// TIA Portal V17 export
// export: Created 2022-07-20T07:01:33.4482737Z, ExportSetting WithDefaults, DisplayName Totally Integrated Automation Portal, DisplayVersion V17, DisplayName TIA Portal Openness, DisplayVersion V17, DisplayName TIA Portal Version Control Interface, DisplayVersion V17, DisplayName SINAMICS Startdrive Advanced, DisplayVersion V17, DisplayName SINAMICS Startdrive G130, G150, S120, S150, SINAMICS MV, S210, DisplayVersion V17, DisplayName SINAMICS Startdrive G110M, G120, G120C, G120D, G120P, G115D, DisplayVersion V17, DisplayName STEP 7 Professional, DisplayVersion V17, DisplayName STEP 7 Safety, DisplayVersion V17, DisplayName WinCC Advanced, DisplayVersion V17
FUNCTION_BLOCK "FB10322_PrinterCompactInkCircuit"   // FB10322, LAD
{ S7_Optimized_Access := 'TRUE' }
VERSION : 0.1
// stored: AutoNumber false, IsIECCheckEnabled false, IsRetainMemResEnabled false, MemoryReserve 100, SetENOAutomatically false, UDAEnableTagReadback false
   VAR_INPUT
      InkWeighScale_RawValue : Int;
      InkWeighScale_CalibrationValue_1 : Real;
      InkWeighScale_CalibrationValue_2 : Real;
      InkWeighScale_HighErrorThreshold : Real;
      InkWeighScale_HighWarningThreshold : Real;
      InkWeighScale_LowWarningThreshold : Real;
      InkWeighScale_LowErrorThreshold : Real;
      InkCircuit_GeneralTankLowLevelSensor : Bool;
      InkCircuit_GeneralTankHighLevelSensor : Bool;
      InkCircuit_SecondaryTankRisingVarnishSensor_B1 : Bool;
      InkCircuit_SecondaryTankRisingVarnishSensor_B2 : Bool;
      InkCircuit_SecondaryTankHighLevelSensor_B1 : Bool;
      InkCircuit_SecondaryTankHighLevelSensor_B2 : Bool;
      WasteWeighScale_RawValue : Int;
      WasteWeighScale_CalibrationValue_1 : Real;
      WasteWeighScale_CalibrationValue_2 : Real;
      WasteWeighScale_HighErrorThreshold : Real;
      WasteWeighScale_HighWarningThreshold : Real;
      WasteWeighScale_LowWarningThreshold : Real;
      WasteWeighScale_LowErrorThreshold : Real;
      FlushWeighScale_RawValue : Int;
      FlushWeighScale_CalibrationValue_1 : Real;
      FlushWeighScale_CalibrationValue_2 : Real;
      FlushWeighScale_HighErrorThreshold : Real;
      FlushWeighScale_HighWarningThreshold : Real;
      FlushWeighScale_LowWarningThreshold : Real;
      FlushWeighScale_LowErrorThreshold : Real;
   END_VAR
   VAR_OUTPUT
      InkWeighScale_SensorCalibrated : Bool;
      InkWeighScale_CalibrationStatus_1 : Bool;
      InkWeighScale_CalibrationStatus_2 : Bool;
      InkWeigh_Scale_ActualValue : Real;
      "InkWeigh_Scale_ActualValue_%" : Real;
      InkWeigh_Scale_HighErrorThresholdReached : Bool;
      InkWeigh_Scale_HighWarningThresholdReached : Bool;
      InkWeigh_Scale_LowWarningThresholdReached : Bool;
      InkWeigh_Scale_LowErrorThresholdReached : Bool;
      InkCircuit_GeneralPump : Bool;
      InkCircuit_SecondaryPump : Bool;
      InkCircuit_GeneralSolenoidValve : Bool;
      InkCircuit_SecondarySolenoidValve_B1 : Bool;
      InkCircuit_SecondarySolenoidValve_B2 : Bool;
      WasteWeighScale_SensorCalibrated : Bool;
      WasteWeighScale_CalibrationStatus_1 : Bool;
      WasteWeighScale_CalibrationStatus_2 : Bool;
      WasteWeigh_Scale_ActualValue : Real;
      "WasteWeigh_Scale_ActualValue_%" : Real;
      WasteWeigh_Scale_HighErrorThresholdReached : Bool;
      WasteWeigh_Scale_HighWarningThresholdReached : Bool;
      WasteWeigh_Scale_LowWarningThresholdReached : Bool;
      WasteWeigh_Scale_LowErrorThresholdReached : Bool;
      FlushWeighScale_SensorCalibrated : Bool;
      FlushWeighScale_CalibrationStatus_1 : Bool;
      FlushWeighScale_CalibrationStatus_2 : Bool;
      FlushWeigh_Scale_ActualValue : Real;
      "FlushWeigh_Scale_ActualValue_%" : Real;
      FlushWeigh_Scale_HighErrorThresholdReached : Bool;
      FlushWeigh_Scale_HighWarningThresholdReached : Bool;
      FlushWeigh_Scale_LowWarningThresholdReached : Bool;
      FlushWeigh_Scale_LowErrorThresholdReached : Bool;
   END_VAR
   VAR_IN_OUT
      InkWeighScale_CalibrationDataX_1 : Real;
      InkWeighScale_CalibrationDataY_1 : Real;
      InkWeighScale_CalibrationDataX_2 : Real;
      InkWeighScale_CalibrationDataY_2 : Real;
      InkWeighScale_RequestCalibration_1 : Bool;
      InkWeighScale_RequestCalibration_2 : Bool;
      InkWeighScale_RequestResetCalibration : Bool;
      InkCircuitRequestAutoregulation : Bool;
      InkCircuitRequestPrincipalFillingTank : Bool;
      InkCircuitRequestSecondaryFillingTank : Bool;
      WasteWeighScale_RequestCalibration_1 : Bool;
      WasteWeighScale_RequestCalibration_2 : Bool;
      WasteWeighScale_RequestResetCalibration : Bool;
      WasteWeighScale_CalibrationDataX_1 : Real;
      WasteWeighScale_CalibrationDataY_1 : Real;
      WasteWeighScale_CalibrationDataX_2 : Real;
      WasteWeighScale_CalibrationDataY_2 : Real;
      FlushWeighScale_CalibrationDataX_1 : Real;
      FlushWeighScale_CalibrationDataY_1 : Real;
      FlushWeighScale_CalibrationDataX_2 : Real;
      FlushWeighScale_CalibrationDataY_2 : Real;
      FlushWeighScale_RequestCalibration_1 : Bool;
      FlushWeighScale_RequestCalibration_2 : Bool;
      FlushWeighScale_RequestResetCalibration : Bool;
   END_VAR
   VAR
      FillingTanksAutoRegulationStateDiagram : Int;
      FB10030_AnalogicalSensor_Instance { S7_SetPoint := 'True'} : "FB10030_AnalogicalSensor";
      R_TRIG_RequestAutoRegulation { S7_SetPoint := 'True'} : R_TRIG;
      F_TRIG_RequestAutoRegulation { S7_SetPoint := 'True'} : F_TRIG;
      R_TRIG_RequestPrincipalFillingTank { S7_SetPoint := 'True'} : R_TRIG;
      F_TRIG_RequestPrincipalFillingTank { S7_SetPoint := 'True'} : F_TRIG;
      R_TRIG_RequestSecondaryFillingTank { S7_SetPoint := 'True'} : R_TRIG;
      F_TRIG_RequestSecondaryFillingTank { S7_SetPoint := 'True'} : F_TRIG;
      FB10030_AnalogicalSensor_Ink { S7_SetPoint := 'True'} : "FB10030_AnalogicalSensor";
      FB10030_AnalogicalSensor_Waste { S7_SetPoint := 'True'} : "FB10030_AnalogicalSensor";
      FB10030_AnalogicalSensor_Flush { S7_SetPoint := 'True'} : "FB10030_AnalogicalSensor";
   END_VAR
   VAR CONSTANT
      "0_WAIT_FOR_AUTOREGULATION_REQUEST" : Int;
      "10_AUTOREGULATION_FILLING_TANKS" : Int := 10;
      "20_PRINCIPAL_FILLING_TANKS" : Int := 20;
      "30_SECONDARY_FILLING_TANKS" : Int := 30;
      "10000_AUTOREGULATION_DONE" : Int := 10000;
   END_VAR
BEGIN

REGION Network 1 (SCL): FirstScan
   IF "FirstScan" THEN
       ;
   END_IF;
END_REGION

REGION Network 2 (SCL): Edge Signal & Timers
   REGION EDGE SIGNAL
       #R_TRIG_RequestAutoRegulation(CLK := #InkCircuitRequestAutoregulation);
       #F_TRIG_RequestAutoRegulation(CLK := #InkCircuitRequestAutoregulation);
       #R_TRIG_RequestPrincipalFillingTank(CLK := #InkCircuitRequestPrincipalFillingTank);
       #F_TRIG_RequestPrincipalFillingTank(CLK := #InkCircuitRequestPrincipalFillingTank);
       #R_TRIG_RequestSecondaryFillingTank(CLK := #InkCircuitRequestSecondaryFillingTank);
       #F_TRIG_RequestSecondaryFillingTank(CLK := #InkCircuitRequestSecondaryFillingTank);
   END_REGION
END_REGION

REGION Network 3 (SCL): Ink Circuit Statement Management
END_REGION

REGION Network 4 (SCL): Ink Circuit Management
   CASE #FillingTanksAutoRegulationStateDiagram OF

       #"0_WAIT_FOR_AUTOREGULATION_REQUEST" :
           #InkCircuit_SecondaryPump := FALSE;
           #InkCircuit_SecondarySolenoidValve_B1 := FALSE;
           #InkCircuit_SecondarySolenoidValve_B2 := FALSE;
           IF #R_TRIG_RequestAutoRegulation.Q THEN
               #FillingTanksAutoRegulationStateDiagram := #"10_AUTOREGULATION_FILLING_TANKS";
           ELSIF #R_TRIG_RequestPrincipalFillingTank.Q THEN
               #FillingTanksAutoRegulationStateDiagram := #"20_PRINCIPAL_FILLING_TANKS";
           ELSIF #R_TRIG_RequestSecondaryFillingTank.Q THEN
               #FillingTanksAutoRegulationStateDiagram := #"30_SECONDARY_FILLING_TANKS";
           END_IF;

       #"10_AUTOREGULATION_FILLING_TANKS" :

           IF  #InkCircuit_GeneralTankHighLevelSensor THEN
               #InkCircuit_GeneralPump := TRUE;
               #InkCircuit_GeneralSolenoidValve := TRUE;
           ELSE
               #InkCircuit_GeneralPump := FALSE;
               #InkCircuit_GeneralSolenoidValve := FALSE;
           END_IF;

           IF #InkCircuit_GeneralTankLowLevelSensor THEN
               #InkCircuit_GeneralPump := TRUE;
               #InkCircuit_GeneralSolenoidValve := TRUE;
               #InkCircuit_SecondaryPump := FALSE; 
               #InkCircuit_SecondarySolenoidValve_B1 := FALSE;
               #InkCircuit_SecondarySolenoidValve_B2 := FALSE;
           END_IF;

           IF NOT #InkCircuit_GeneralTankLowLevelSensor THEN
               IF  #InkCircuit_SecondaryTankHighLevelSensor_B1 AND #InkCircuit_SecondaryTankHighLevelSensor_B2 THEN
                   #InkCircuit_SecondaryPump := TRUE;
                   #InkCircuit_SecondarySolenoidValve_B1 := TRUE;
                   #InkCircuit_SecondarySolenoidValve_B2 := TRUE;
               ELSIF #InkCircuit_SecondaryTankHighLevelSensor_B2 THEN
                   #InkCircuit_SecondaryPump := TRUE;
                   #InkCircuit_SecondarySolenoidValve_B2 := TRUE; 
                   #InkCircuit_SecondarySolenoidValve_B1 := FALSE;
               ELSIF #InkCircuit_SecondaryTankHighLevelSensor_B1 THEN
                   #InkCircuit_SecondaryPump := TRUE;
                   #InkCircuit_SecondarySolenoidValve_B1 := TRUE;
                   #InkCircuit_SecondarySolenoidValve_B2 := FALSE;
               ELSE
                   #InkCircuit_SecondaryPump := FALSE;
                   #InkCircuit_SecondarySolenoidValve_B1 := FALSE;
                   #InkCircuit_SecondarySolenoidValve_B2 := FALSE;
               END_IF;
           END_IF;

           ////////////////////////////////////////////////////////////////
           IF #F_TRIG_RequestAutoRegulation.Q THEN
               #FillingTanksAutoRegulationStateDiagram := #"10000_AUTOREGULATION_DONE";
           END_IF;


       #"20_PRINCIPAL_FILLING_TANKS" :

           IF  #InkCircuit_GeneralTankHighLevelSensor THEN
               #InkCircuit_GeneralPump := TRUE;
               #InkCircuit_GeneralSolenoidValve := TRUE;
           ELSE
               #InkCircuit_GeneralPump := FALSE;
               #InkCircuit_GeneralSolenoidValve := FALSE;
           END_IF;

           IF #F_TRIG_RequestAutoRegulation.Q THEN
               #FillingTanksAutoRegulationStateDiagram := #"10000_AUTOREGULATION_DONE";
           END_IF;


           ////////////////////////////////////////////////////////////////
           IF #F_TRIG_RequestPrincipalFillingTank.Q THEN
               #FillingTanksAutoRegulationStateDiagram := #"10000_AUTOREGULATION_DONE";
           END_IF;


       #"30_SECONDARY_FILLING_TANKS":

           IF NOT #InkCircuit_GeneralTankLowLevelSensor THEN
               IF  #InkCircuit_SecondaryTankHighLevelSensor_B1 AND #InkCircuit_SecondaryTankHighLevelSensor_B2 THEN
                   #InkCircuit_SecondaryPump := TRUE;
                   #InkCircuit_SecondarySolenoidValve_B1 := TRUE;
                   #InkCircuit_SecondarySolenoidValve_B2 := TRUE;
               ELSIF #InkCircuit_SecondaryTankHighLevelSensor_B2 THEN
                   #InkCircuit_SecondaryPump := TRUE;
                   #InkCircuit_SecondarySolenoidValve_B2 := TRUE;
                   #InkCircuit_SecondarySolenoidValve_B1 := FALSE;
               ELSIF  #InkCircuit_SecondaryTankHighLevelSensor_B1 THEN
                   #InkCircuit_SecondaryPump := TRUE;
                   #InkCircuit_SecondarySolenoidValve_B1 := TRUE;
                   #InkCircuit_SecondarySolenoidValve_B2 := FALSE;
               ELSE
                   #InkCircuit_SecondaryPump := FALSE;
                   #InkCircuit_SecondarySolenoidValve_B1 := FALSE;
                   #InkCircuit_SecondarySolenoidValve_B2 := FALSE;
               END_IF;
           END_IF;



           ////////////////////////////////////////////////////////////////
           IF #F_TRIG_RequestSecondaryFillingTank.Q THEN
               #FillingTanksAutoRegulationStateDiagram := #"10000_AUTOREGULATION_DONE";
           END_IF;

       #"10000_AUTOREGULATION_DONE":
           #InkCircuit_GeneralPump := FALSE;
           #InkCircuit_GeneralSolenoidValve := FALSE;
           #InkCircuit_SecondaryPump := FALSE;
           #InkCircuit_SecondarySolenoidValve_B1 := FALSE;
           #InkCircuit_SecondarySolenoidValve_B2 := FALSE;
           #FillingTanksAutoRegulationStateDiagram := #"0_WAIT_FOR_AUTOREGULATION_REQUEST";
   END_CASE;
END_REGION

REGION Network 5 (SCL): Ink Circuit State Management
END_REGION

REGION Network 6: Ink Weigh Scales Management
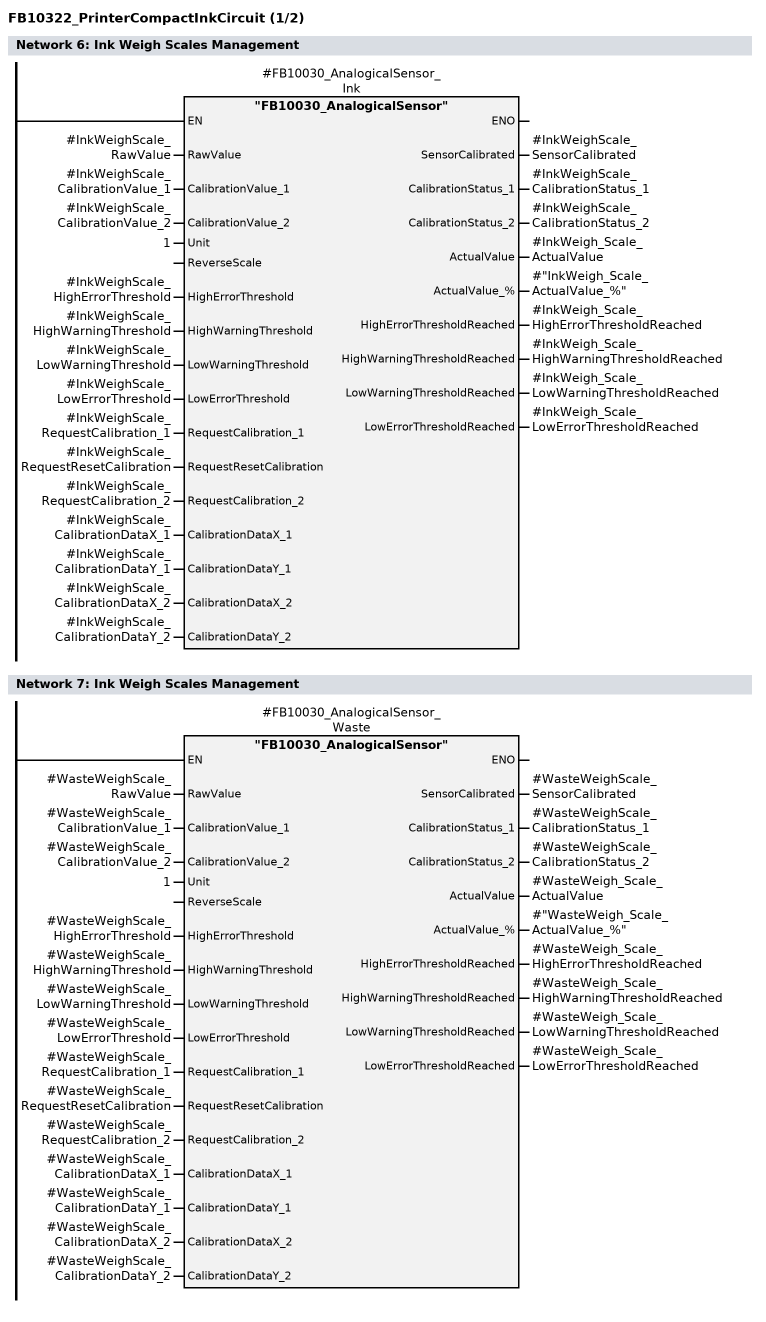
   RUNG wire#powerrail
      #FB10030_AnalogicalSensor_Ink(RawValue := #InkWeighScale_RawValue, CalibrationValue_1 := #InkWeighScale_CalibrationValue_1, CalibrationValue_2 := #InkWeighScale_CalibrationValue_2, Unit := 1, ReverseScale :=, HighErrorThreshold := #InkWeighScale_HighErrorThreshold, HighWarningThreshold := #InkWeighScale_HighWarningThreshold, LowWarningThreshold := #InkWeighScale_LowWarningThreshold, LowErrorThreshold := #InkWeighScale_LowErrorThreshold, RequestCalibration_1 := #InkWeighScale_RequestCalibration_1, RequestResetCalibration := #InkWeighScale_RequestResetCalibration, RequestCalibration_2 := #InkWeighScale_RequestCalibration_2, CalibrationDataX_1 := #InkWeighScale_CalibrationDataX_1, CalibrationDataY_1 := #InkWeighScale_CalibrationDataY_1, CalibrationDataX_2 := #InkWeighScale_CalibrationDataX_2, CalibrationDataY_2 := #InkWeighScale_CalibrationDataY_2, SensorCalibrated => #InkWeighScale_SensorCalibrated, CalibrationStatus_1 => #InkWeighScale_CalibrationStatus_1, CalibrationStatus_2 => #InkWeighScale_CalibrationStatus_2, ActualValue => #InkWeigh_Scale_ActualValue, "ActualValue_%" => #"InkWeigh_Scale_ActualValue_%", HighErrorThresholdReached => #InkWeigh_Scale_HighErrorThresholdReached, HighWarningThresholdReached => #InkWeigh_Scale_HighWarningThresholdReached, LowWarningThresholdReached => #InkWeigh_Scale_LowWarningThresholdReached, LowErrorThresholdReached => #InkWeigh_Scale_LowErrorThresholdReached)
   END_RUNG
   // the same network as SCL:
   #FB10030_AnalogicalSensor_Ink(RawValue := #InkWeighScale_RawValue,   // "FB10030_AnalogicalSensor"
                           CalibrationValue_1 := #InkWeighScale_CalibrationValue_1,
                           CalibrationValue_2 := #InkWeighScale_CalibrationValue_2,
                           Unit := 1,
                           HighErrorThreshold := #InkWeighScale_HighErrorThreshold,
                           HighWarningThreshold := #InkWeighScale_HighWarningThreshold,
                           LowWarningThreshold := #InkWeighScale_LowWarningThreshold,
                           LowErrorThreshold := #InkWeighScale_LowErrorThreshold,
                           RequestCalibration_1 := #InkWeighScale_RequestCalibration_1,
                           RequestResetCalibration := #InkWeighScale_RequestResetCalibration,
                           RequestCalibration_2 := #InkWeighScale_RequestCalibration_2,
                           CalibrationDataX_1 := #InkWeighScale_CalibrationDataX_1,
                           CalibrationDataY_1 := #InkWeighScale_CalibrationDataY_1,
                           CalibrationDataX_2 := #InkWeighScale_CalibrationDataX_2,
                           CalibrationDataY_2 := #InkWeighScale_CalibrationDataY_2,
                           SensorCalibrated => #InkWeighScale_SensorCalibrated,
                           CalibrationStatus_1 => #InkWeighScale_CalibrationStatus_1,
                           CalibrationStatus_2 => #InkWeighScale_CalibrationStatus_2,
                           ActualValue => #InkWeigh_Scale_ActualValue,
                           "ActualValue_%" => #"InkWeigh_Scale_ActualValue_%",
                           HighErrorThresholdReached => #InkWeigh_Scale_HighErrorThresholdReached,
                           HighWarningThresholdReached => #InkWeigh_Scale_HighWarningThresholdReached,
                           LowWarningThresholdReached => #InkWeigh_Scale_LowWarningThresholdReached,
                           LowErrorThresholdReached => #InkWeigh_Scale_LowErrorThresholdReached);
END_REGION

REGION Network 7: Ink Weigh Scales Management
   RUNG wire#powerrail
      #FB10030_AnalogicalSensor_Waste(RawValue := #WasteWeighScale_RawValue, CalibrationValue_1 := #WasteWeighScale_CalibrationValue_1, CalibrationValue_2 := #WasteWeighScale_CalibrationValue_2, Unit := 1, HighErrorThreshold := #WasteWeighScale_HighErrorThreshold, HighWarningThreshold := #WasteWeighScale_HighWarningThreshold, LowWarningThreshold := #WasteWeighScale_LowWarningThreshold, LowErrorThreshold := #WasteWeighScale_LowErrorThreshold, RequestCalibration_1 := #WasteWeighScale_RequestCalibration_1, RequestCalibration_2 := #WasteWeighScale_RequestCalibration_2, RequestResetCalibration := #WasteWeighScale_RequestResetCalibration, CalibrationDataX_1 := #WasteWeighScale_CalibrationDataX_1, CalibrationDataY_1 := #WasteWeighScale_CalibrationDataY_1, CalibrationDataX_2 := #WasteWeighScale_CalibrationDataX_2, CalibrationDataY_2 := #WasteWeighScale_CalibrationDataY_2, SensorCalibrated => #WasteWeighScale_SensorCalibrated, CalibrationStatus_1 => #WasteWeighScale_CalibrationStatus_1, CalibrationStatus_2 => #WasteWeighScale_CalibrationStatus_2, ActualValue => #WasteWeigh_Scale_ActualValue, "ActualValue_%" => #"WasteWeigh_Scale_ActualValue_%", HighErrorThresholdReached => #WasteWeigh_Scale_HighErrorThresholdReached, HighWarningThresholdReached => #WasteWeigh_Scale_HighWarningThresholdReached, LowWarningThresholdReached => #WasteWeigh_Scale_LowWarningThresholdReached, LowErrorThresholdReached => #WasteWeigh_Scale_LowErrorThresholdReached, ReverseScale :=)
   END_RUNG
   // the same network as SCL:
   #FB10030_AnalogicalSensor_Waste(RawValue := #WasteWeighScale_RawValue,   // "FB10030_AnalogicalSensor"
                           CalibrationValue_1 := #WasteWeighScale_CalibrationValue_1,
                           CalibrationValue_2 := #WasteWeighScale_CalibrationValue_2,
                           Unit := 1,
                           HighErrorThreshold := #WasteWeighScale_HighErrorThreshold,
                           HighWarningThreshold := #WasteWeighScale_HighWarningThreshold,
                           LowWarningThreshold := #WasteWeighScale_LowWarningThreshold,
                           LowErrorThreshold := #WasteWeighScale_LowErrorThreshold,
                           RequestCalibration_1 := #WasteWeighScale_RequestCalibration_1,
                           RequestResetCalibration := #WasteWeighScale_RequestResetCalibration,
                           RequestCalibration_2 := #WasteWeighScale_RequestCalibration_2,
                           CalibrationDataX_1 := #WasteWeighScale_CalibrationDataX_1,
                           CalibrationDataY_1 := #WasteWeighScale_CalibrationDataY_1,
                           CalibrationDataX_2 := #WasteWeighScale_CalibrationDataX_2,
                           CalibrationDataY_2 := #WasteWeighScale_CalibrationDataY_2,
                           SensorCalibrated => #WasteWeighScale_SensorCalibrated,
                           CalibrationStatus_1 => #WasteWeighScale_CalibrationStatus_1,
                           CalibrationStatus_2 => #WasteWeighScale_CalibrationStatus_2,
                           ActualValue => #WasteWeigh_Scale_ActualValue,
                           "ActualValue_%" => #"WasteWeigh_Scale_ActualValue_%",
                           HighErrorThresholdReached => #WasteWeigh_Scale_HighErrorThresholdReached,
                           HighWarningThresholdReached => #WasteWeigh_Scale_HighWarningThresholdReached,
                           LowWarningThresholdReached => #WasteWeigh_Scale_LowWarningThresholdReached,
                           LowErrorThresholdReached => #WasteWeigh_Scale_LowErrorThresholdReached);
END_REGION

REGION Network 9: Ink Weigh Scales Management
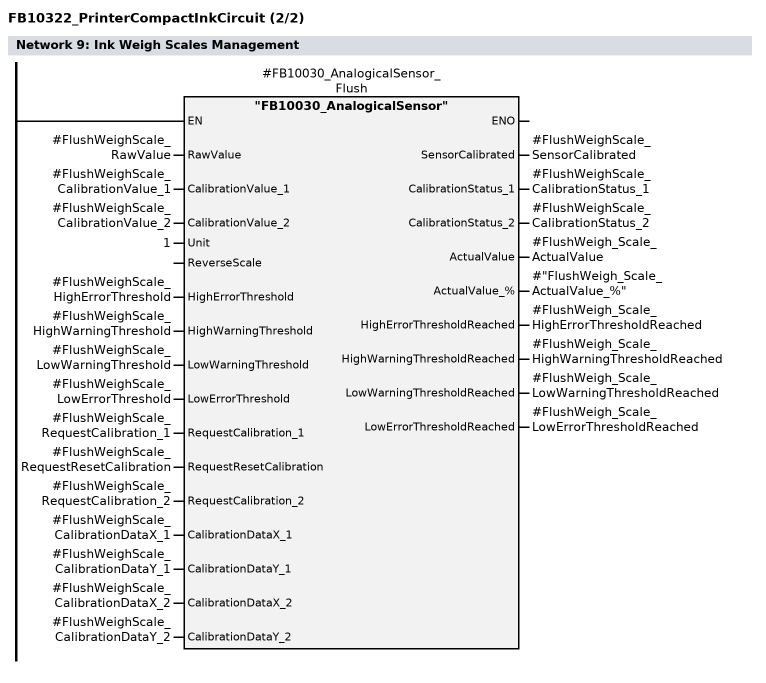
   RUNG wire#powerrail
      #FB10030_AnalogicalSensor_Flush(RawValue := #FlushWeighScale_RawValue, CalibrationValue_1 := #FlushWeighScale_CalibrationValue_1, CalibrationValue_2 := #FlushWeighScale_CalibrationValue_2, Unit := 1, HighErrorThreshold := #FlushWeighScale_HighErrorThreshold, HighWarningThreshold := #FlushWeighScale_HighWarningThreshold, LowWarningThreshold := #FlushWeighScale_LowWarningThreshold, LowErrorThreshold := #FlushWeighScale_LowErrorThreshold, RequestCalibration_1 := #FlushWeighScale_RequestCalibration_1, RequestCalibration_2 := #FlushWeighScale_RequestCalibration_2, RequestResetCalibration := #FlushWeighScale_RequestResetCalibration, CalibrationDataX_1 := #FlushWeighScale_CalibrationDataX_1, CalibrationDataY_1 := #FlushWeighScale_CalibrationDataY_1, CalibrationDataX_2 := #FlushWeighScale_CalibrationDataX_2, CalibrationDataY_2 := #FlushWeighScale_CalibrationDataY_2, SensorCalibrated => #FlushWeighScale_SensorCalibrated, CalibrationStatus_1 => #FlushWeighScale_CalibrationStatus_1, CalibrationStatus_2 => #FlushWeighScale_CalibrationStatus_2, ActualValue => #FlushWeigh_Scale_ActualValue, "ActualValue_%" => #"FlushWeigh_Scale_ActualValue_%", HighErrorThresholdReached => #FlushWeigh_Scale_HighErrorThresholdReached, HighWarningThresholdReached => #FlushWeigh_Scale_HighWarningThresholdReached, LowWarningThresholdReached => #FlushWeigh_Scale_LowWarningThresholdReached, LowErrorThresholdReached => #FlushWeigh_Scale_LowErrorThresholdReached, ReverseScale :=)
   END_RUNG
   // the same network as SCL:
   #FB10030_AnalogicalSensor_Flush(RawValue := #FlushWeighScale_RawValue,   // "FB10030_AnalogicalSensor"
                           CalibrationValue_1 := #FlushWeighScale_CalibrationValue_1,
                           CalibrationValue_2 := #FlushWeighScale_CalibrationValue_2,
                           Unit := 1,
                           HighErrorThreshold := #FlushWeighScale_HighErrorThreshold,
                           HighWarningThreshold := #FlushWeighScale_HighWarningThreshold,
                           LowWarningThreshold := #FlushWeighScale_LowWarningThreshold,
                           LowErrorThreshold := #FlushWeighScale_LowErrorThreshold,
                           RequestCalibration_1 := #FlushWeighScale_RequestCalibration_1,
                           RequestResetCalibration := #FlushWeighScale_RequestResetCalibration,
                           RequestCalibration_2 := #FlushWeighScale_RequestCalibration_2,
                           CalibrationDataX_1 := #FlushWeighScale_CalibrationDataX_1,
                           CalibrationDataY_1 := #FlushWeighScale_CalibrationDataY_1,
                           CalibrationDataX_2 := #FlushWeighScale_CalibrationDataX_2,
                           CalibrationDataY_2 := #FlushWeighScale_CalibrationDataY_2,
                           SensorCalibrated => #FlushWeighScale_SensorCalibrated,
                           CalibrationStatus_1 => #FlushWeighScale_CalibrationStatus_1,
                           CalibrationStatus_2 => #FlushWeighScale_CalibrationStatus_2,
                           ActualValue => #FlushWeigh_Scale_ActualValue,
                           "ActualValue_%" => #"FlushWeigh_Scale_ActualValue_%",
                           HighErrorThresholdReached => #FlushWeigh_Scale_HighErrorThresholdReached,
                           HighWarningThresholdReached => #FlushWeigh_Scale_HighWarningThresholdReached,
                           LowWarningThresholdReached => #FlushWeigh_Scale_LowWarningThresholdReached,
                           LowErrorThresholdReached => #FlushWeigh_Scale_LowErrorThresholdReached);
END_REGION
END_FUNCTION_BLOCK
